stInitData.ModelParameters.filter_tau_slow_T_1[2] := 0.00079577471545947667;
stInitData.ModelParameters.filter_tau_slow_T_1[3] := 0.00079577471545947667;
stInitData.ModelParameters.filter_tau_slow_T_1[4] := 0.00079577471545947667;
stInitData.ModelParameters.filter_tau_slow_T_1[5] := 0.00079577471545947667;
stInitData.ModelParameters.filter_tau_slow_T_1[6] := 0.00079577471545947667;
stInitData.ModelParameters.filter_theta_p_slow_T_1[0] := 0.00079577471545947667;
stInitData.ModelParameters.filter_theta_p_slow_T_1[1] := 0.00079577471545947667;
stInitData.ModelParameters.filter_theta_p_slow_T_1[2] := 0.00079577471545947667;
stInitData.ModelParameters.filter_theta_p_slow_T_1[3] := 0.00079577471545947667;
stInitData.ModelParameters.filter_theta_p_slow_T_1[4] := 0.00079577471545947667;
stInitData.ModelParameters.filter_theta_p_slow_T_1[5] := 0.00079577471545947667;
stInitData.ModelParameters.filter_theta_p_slow_T_1[6] := 0.00079577471545947667;
stInitData.ModelParameters.filter_theta_slow_T_1[0] := 0.00079577471545947667;
stInitData.ModelParameters.filter_theta_slow_T_1[1] := 0.00079577471545947667;
stInitData.ModelParameters.filter_theta_slow_T_1[2] := 0.00079577471545947667;
stInitData.ModelParameters.filter_theta_slow_T_1[3] := 0.00079577471545947667;
stInitData.ModelParameters.filter_theta_slow_T_1[4] := 0.00079577471545947667;
stInitData.ModelParameters.filter_theta_slow_T_1[5] := 0.00079577471545947667;
stInitData.ModelParameters.filter_theta_slow_T_1[6] := 0.00079577471545947667;
stInitData.ModelParameters.height_of_catch := 0.90000000000000002;
stInitData.ModelParameters.sensor_torque_offset[0] := 0.53000000000000003;
stInitData.ModelParameters.sensor_torque_offset[1] := -0.095000000000000001;
stInitData.ModelParameters.sensor_torque_offset[2] := -0.189;
stInitData.ModelParameters.sensor_torque_offset[3] := 0.070000000000000007;
stInitData.ModelParameters.sensor_torque_offset[4] := -0.058000000000000003;
stInitData.ModelParameters.sensor_torque_offset[5] := 0.0025000000000000001;
stInitData.ModelParameters.sensor_torque_offset[6] := -0.12;
stInitData.ModelParameters.Constant21_Value := 0;
stInitData.ModelParameters.Constant19_Value := 1;
stInitData.ModelParameters.pd_Y0 := 0;
stInitData.ModelParameters.pd_p_Y0 := 0;
stInitData.ModelParameters.t_catch_pred_Y0 := 0;
stInitData.ModelParameters.use_pred_Y0 := 0;
stInitData.ModelParameters.pred_update_Y0 := 0;
stInitData.ModelParameters.Throw_Constant_Value := 0;
stInitData.ModelParameters.Constant25_Value := -0.080000000000000002;
stInitData.ModelParameters.Constant26_Value := -0.10000000000000001;
stInitData.ModelParameters.Constant30_Value := 0;
stInitData.ModelParameters.Constant27_Value := 0;
stInitData.ModelParameters.Constant28_Value := 0;
stInitData.ModelParameters.Constant29_Value := 0;
stInitData.ModelParameters.Constant1_Value := 3.6000000000000001;
stInitData.ModelParameters.Constant17_Value := 0;
stInitData.ModelParameters.Constant_Value := 100;
stInitData.ModelParameters.Constant4_Value[0] := 0.40000000000000002;
stInitData.ModelParameters.Constant4_Value[1] := 0;
stInitData.ModelParameters.Constant4_Value[2] := 0.69999999999999996;
stInitData.ModelParameters.Constant2_Value := 100;
stInitData.ModelParameters.Constant3_Value := 0;
stInitData.ModelParameters.Constant18_Value := 5;
stInitData.ModelParameters.MotionEnableValue_Value := 0;
stInitData.ModelParameters.MotionDisableValue_Value := 0;
stInitData.ModelParameters.RigidBodyControllerSelector_Value := 2;
stInitData.ModelParameters.ManualSwitch2_CurrentSetting := 0;
stInitData.ModelParameters.ManualSwitch7_CurrentSetting := 0;
stInitData.ContextInfoArr_0_TaskOidHdr.indexGroup := 0;
stInitData.ContextInfoArr_0_TaskOidHdr.indexOffset := 16#03002060;
stInitData.ContextInfoArr_0_TaskOidHdr.cbData := SIZEOF(stInitData.ContextInfoArr_0_TaskOid);
stInitData.ContextInfoArr_0_TaskPriorityHdr.indexGroup := 0;
stInitData.ContextInfoArr_0_TaskPriorityHdr.indexOffset := 16#03002070;
stInitData.ContextInfoArr_0_TaskPriorityHdr.cbData := SIZEOF(stInitData.ContextInfoArr_0_TaskPriority);
stInitData.ContextInfoArr_0_TaskCycleTimeNsHdr.indexGroup := 0;
stInitData.ContextInfoArr_0_TaskCycleTimeNsHdr.indexOffset := 16#03002080;
stInitData.ContextInfoArr_0_TaskCycleTimeNsHdr.cbData := SIZEOF(stInitData.ContextInfoArr_0_TaskCycleTimeNs);
stInitData.ContextInfoArr_0_TaskPortHdr.indexGroup := 0;
stInitData.ContextInfoArr_0_TaskPortHdr.indexOffset := 16#03002090;
stInitData.ContextInfoArr_0_TaskPortHdr.cbData := SIZEOF(stInitData.ContextInfoArr_0_TaskPort);
stInitData.ContextInfoArr_0_TaskSortOrderHdr.indexGroup := 0;
stInitData.ContextInfoArr_0_TaskSortOrderHdr.indexOffset := 16#030020b0;
stInitData.ContextInfoArr_0_TaskSortOrderHdr.cbData := SIZEOF(stInitData.ContextInfoArr_0_TaskSortOrder);
stInitData.Header.cbData := SIZEOF(stInitData)-SIZEOF(stInitData.Header);
stInitData.Header.uiElmCnt := 11;


// set pointer to InitData structure
SetInitDataInfo(ADR(stInitData));

// set DataArea information
SetDataAreaInfo(ADR(arrDataAreas),2);
arrDataAreas[1].nDataAreaId := 0;
arrDataAreas[1].nSize := SIZEOF(stInput);
arrDataAreas[1].pPlcVar := ADR(stInput);
arrDataAreas[1].pModuleProcImg := 0;
arrDataAreas[1].eDataAreaType := E_TcMatSimDataAreaType.InputDst;
arrDataAreas[2].nDataAreaId := 1;
arrDataAreas[2].nSize := SIZEOF(stOutput);
arrDataAreas[2].pPlcVar := ADR(stOutput);
arrDataAreas[2].pModuleProcImg := 0;
arrDataAreas[2].eDataAreaType := E_TcMatSimDataAreaType.OutputSrc;


// initialize basic interface pointers and return
FB_init := SUCCEEDED(Init(oid));
                  
                
END_METHOD

METHOD Execute : HRESULT
                  
IF (SUCCEEDED(hResult)) THEN
  hResult := VerifyParameters();
END_IF

// update DataArea information
SetDataAreaInfo(ADR(arrDataAreas),2);
arrDataAreas[1].nDataAreaId := 0;
arrDataAreas[1].nSize := SIZEOF(stInput);
arrDataAreas[1].pPlcVar := ADR(stInput);
arrDataAreas[1].pModuleProcImg := 0;
arrDataAreas[1].eDataAreaType := E_TcMatSimDataAreaType.InputDst;
arrDataAreas[2].nDataAreaId := 1;
arrDataAreas[2].nSize := SIZEOF(stOutput);
arrDataAreas[2].pPlcVar := ADR(stOutput);
arrDataAreas[2].pModuleProcImg := 0;
arrDataAreas[2].eDataAreaType := E_TcMatSimDataAreaType.OutputSrc;

	
// call base method
Execute := SUPER^.Execute();
                  
                
END_METHOD

{attribute 'object_name' := 'VerifyParameters'}
METHOD VerifyParameters : HRESULT
  VAR
    moduleCallByParam : TctModuleCallByType;
  END_VAR
                  
IF (bParametersVerified) THEN
  VerifyParameters := Tc2_System.E_HRESULTAdsErr.HRESULT_ADS_NOERROR;
ELSE
  VerifyParameters := GetObjPara(stInitData.CallByHdr.indexOffset,SIZEOF(moduleCallByParam),ADR(moduleCallByParam));
  
  // check the "CallBy" parameter to be set to "Module"
  IF (SUCCEEDED(VerifyParameters) AND (moduleCallByParam <> TctModuleCallByType.Module)) THEN
      VerifyParameters := Tc2_System.E_HRESULTAdsErr.INVALIDPARM;
  END_IF
  
  // set the parameters verified flag
  bParametersVerified := SUCCEEDED(VerifyParameters);
END_IF
                  
                
END_METHOD

PROPERTY InitData : ST_controller_ballcatcher_inv_kinInitData
GET
                    InitData := stInitData;
                  
END_GET
SET
                    stInitData := InitData;
                  
END_SET
END_PROPERTY
END_FUNCTION_BLOCK
